Yaskawa INFORM job: OK_R2_O7,1(P)(180,90)OKKR.JBI

/JOB
//NAME OK_R2_O7,1(P)(180,90)OKKR
///FOLDERNAME X4
//POS
///NPOS 170,170,170,10,0,0
///TOOL 0
///POSTYPE PULSE
///PULSE
C00000=-124821,-99493,-112304,-12763,69065,-63689
C00001=-125572,-109805,-73016,-14673,60245,-62954
C00002=-125529,-106474,-67472,-14933,58606,-62713
C00003=-125513,-105112,-65225,-15043,57949,-62613
C00004=-125931,-102761,-62431,-15024,57379,-62697
C00005=-125513,-105112,-65225,-15043,57949,-62613
C00006=-115155,-116372,-68286,-18066,56230,-58210
C00007=-113191,-117815,-68179,-18629,55880,-57359
C00008=-115155,-116372,-68286,-18066,56230,-58210
C00009=-115178,-117983,-70589,-17944,56786,-58316
C00010=-115234,-121991,-76286,-17657,58155,-58571
C00011=-120585,-128453,-93269,-11576,67473,-62203
C00012=-120088,-125588,-88095,-11803,65866,-61858
C00013=-119888,-124404,-86000,-11898,65228,-61718
C00014=-120403,-122095,-83389,-11849,64741,-61858
C00015=-119888,-124404,-86000,-11898,65228,-61718
C00016=-108971,-134765,-87218,-14096,62473,-57335
C00017=-106536,-136286,-87094,-14543,62053,-56368
C00018=-108971,-134765,-87218,-14096,62473,-57335
C00019=-109237,-136316,-89410,-13991,62964,-57496
C00020=-109895,-140195,-94852,-13741,64173,-57891
C00021=-125550,-127827,-102093,-6546,69504,-64123
C00022=-124619,-125212,-97090,-6829,67858,-63692
C00023=-124246,-124117,-95064,-6945,67210,-63518
C00024=-124692,-122258,-93043,-6859,66886,-63662
C00025=-124246,-124117,-95064,-6945,67210,-63518
C00026=-116781,-135280,-96410,-8903,63075,-60474
C00027=-115485,-136646,-96399,-9241,62517,-59943
C00028=-116781,-135280,-96410,-8903,63075,-60474
C00029=-117208,-136830,-98557,-8770,63547,-60670
C00030=-118273,-140721,-103898,-8447,64709,-61154
C00031=-124821,-99493,-112304,-12763,69065,-63689
C00032=-107946,-141846,-124280,-39630,59824,-29939
C00033=-109801,-105651,-82130,-40578,68986,-43153
C00034=-114208,-101668,-58675,-42695,64807,-43138
C00035=-119984,-99571,-57689,-39111,62764,-45440
C00036=-120682,-97946,-55361,-39253,61992,-45447
C00037=-120683,-95917,-52962,-39397,61652,-45306
C00038=-120682,-97946,-55361,-39253,61992,-45447
C00039=-120456,-110188,-58493,-40823,58706,-43930
C00040=-120434,-113010,-58717,-41347,57713,-43467
C00041=-120456,-110188,-58493,-40823,58706,-43930
C00042=-119614,-112042,-60852,-40668,59458,-43865
C00043=-117480,-116658,-66680,-40315,61328,-43677
C00044=-118912,-112770,-80088,-37329,68797,-47272
C00045=-120652,-109018,-74647,-37486,66909,-47352
C00046=-121340,-107497,-72445,-37559,66154,-47379
C00047=-121335,-105659,-70425,-37638,65916,-47288
C00048=-121340,-107497,-72445,-37559,66154,-47379
C00049=-119649,-123976,-76874,-39368,62335,-45109
C00050=-119586,-126928,-76972,-39856,61227,-44619
C00051=-119649,-123976,-76874,-39368,62335,-45109
C00052=-118793,-125859,-79136,-39287,63040,-45003
C00053=-116627,-130595,-84751,-39109,64786,-44716
C00054=-118466,-121522,-88777,-40234,61844,-44303
C00055=-120300,-116165,-83095,-40134,60429,-44594
C00056=-121009,-114063,-80811,-40109,59853,-44695
C00057=-121007,-112566,-79277,-40173,59718,-44636
C00058=-121009,-114063,-80811,-40109,59853,-44695
C00059=-120085,-126490,-82623,-42400,56261,-42581
C00060=-120051,-129243,-82840,-42985,55321,-42099
C00061=-120085,-126490,-82623,-42400,56261,-42581
C00062=-119241,-128903,-84937,-42455,56795,-42402
C00063=-117047,-135114,-90707,-42638,58096,-41900
C00064=-109801,-105651,-82130,-40578,68986,-43153
C00065=-122192,-109712,-75470,-6994,72350,-47586
C00066=-120404,-106593,-70167,-7203,70857,-46871
C00067=-119689,-105303,-68015,-7288,70263,-46584
C00068=-119701,-103141,-65704,-7302,69952,-46569
C00069=-119689,-105303,-68015,-7288,70263,-46584
C00070=-121664,-119459,-71492,-7384,64996,-46952
C00071=-121705,-121620,-70662,-7478,63384,-46863
C00072=-121664,-119459,-71492,-7384,64996,-46952
C00073=-122530,-121046,-73712,-7280,65466,-47290
C00074=-124694,-124965,-79200,-7022,66635,-48130
C00075=-123098,-114349,-89377,-6073,92150,-50670
C00076=-121321,-114367,-85375,-5874,89822,-49955
C00077=-120587,-114243,-83719,-5794,88924,-49665
C00078=-120588,-112592,-81737,-5794,88555,-49647
C00079=-120587,-114243,-83719,-5794,88924,-49665
C00080=-120582,-131484,-87781,-5822,82597,-49371
C00081=-120567,-134184,-87056,-5843,80774,-49281
C00082=-120582,-131484,-87781,-5822,82597,-49371
C00083=-121475,-132061,-89612,-5910,83359,-49704
C00084=-123618,-133239,-94082,-6121,85336,-50515
C00085=-122927,-125261,-102860,-5781,84947,-50274
C00086=-121065,-123842,-98350,-5851,83046,-49551
C00087=-120312,-123169,-96506,-5880,82315,-49259
C00088=-120315,-121628,-95025,-5881,82198,-49255
C00089=-120312,-123169,-96506,-5880,82315,-49259
C00090=-120906,-137774,-98641,-5969,76113,-49167
C00091=-120906,-140631,-98437,-6009,74527,-49089
C00092=-120906,-137774,-98641,-5969,76113,-49167
C00093=-121779,-138951,-100636,-5931,76668,-49494
C00094=-123931,-141761,-105561,-5836,78092,-50300
C00095=-120586,-134579,-103358,-4485,83037,-11114
C00096=-120585,-131353,-98423,-4497,81662,-11065
C00097=-122535,-156833,-100738,-4824,60146,-10922
C00098=-120522,-156760,-100374,-5125,60080,-10181
C00099=-120535,-157089,-102253,-5074,61063,-10231
C00100=-122383,-157140,-100927,-4850,60115,-10864
C00101=-120539,-156480,-102582,-5050,61576,-10256
C00102=-120540,-162054,-108025,-5027,62060,-10277
C00103=-120585,-128403,-93705,-30706,64058,-34634
C00104=-120567,-133478,-88916,-33924,55149,-31719
C00105=-122986,-144654,-84100,-43838,39416,-25487
C00106=-120515,-146044,-85731,-44330,40764,-24767
C00107=-120500,-145449,-83725,-45099,40100,-24310
C00108=-106025,-137078,-79844,-52562,53027,-19025
C00109=-92891,-135829,-78811,-56182,61380,-16538
C00110=-84226,-141246,-87089,-54613,67539,-15724
C00111=-120583,-120823,-82153,-31538,61287,-33793
C00112=-120582,-117425,-76976,-31951,60054,-33402
C00113=-121881,-133792,-71539,-46034,38379,-24018
C00114=-120512,-134879,-73160,-46011,39332,-23778
C00115=-120497,-134214,-71093,-46846,38685,-23292
C00116=-121927,-133795,-71532,-46028,38354,-24030
C00117=-120517,-134657,-73586,-45684,39595,-23969
C00118=-120519,-139446,-79120,-44885,40271,-24439
C00119=-120584,-125271,-89201,-16167,69548,-26657
C00120=-120507,-146022,-83749,-22694,42309,-21504
C00121=-122688,-146060,-81853,-22354,40667,-22120
C00122=-120486,-145618,-81276,-23272,41099,-21150
C00123=-120502,-146316,-83328,-22869,41930,-21396
C00124=-122679,-146211,-81883,-22385,40613,-22104
C00125=-120507,-145977,-83749,-22685,42330,-21510
C00126=-120508,-151207,-89253,-22395,42978,-21687
C00127=-120580,-111726,-68534,-21389,53781,-37532
C00128=-127451,-113025,-63775,-15084,47988,-22225
C00129=-127911,-112838,-61925,-15165,46900,-22250
C00130=-127661,-113044,-61494,-15348,46585,-22086
C00131=-127527,-113364,-63423,-15147,47596,-22194
C00132=-128157,-113633,-62740,-8323,46523,-24870
C00133=-127382,-113593,-64507,-8470,47695,-24640
C00134=-127382,-117368,-69886,-8296,49052,-24759
C00135=-120579,-109195,-64459,-33713,55342,-34372
C00136=-120513,-118310,-53934,-51164,35641,-23385
C00137=-121307,-116964,-51688,-51749,34808,-23220
C00138=-120509,-118473,-53470,-51568,35408,-23161
C00139=-120494,-117670,-51270,-52630,34821,-22576
C00140=-120628,-116889,-51668,-51870,35163,-23019
C00141=-120514,-118344,-53933,-51183,35630,-23374
C00142=-102692,-110233,-56027,-52580,57513,-23173
C00143=-107946,-141846,-124280,-39630,59824,-29939
C00144=-124821,-99493,-112304,-12763,69065,-63689
C00145=-120586,-135028,-103405,-1882,87308,19162
C00146=-95049,-154551,-101030,-14337,69428,29511
C00147=-96126,-153925,-99141,-14396,68431,29253
C00148=-94146,-154571,-100597,-14373,69310,29842
C00149=-92471,-153341,-98557,-14446,68990,30473
C00150=-96000,-153530,-99051,-14384,68596,29277
C00151=-95031,-154583,-101021,-14339,69408,29519
C00152=-95039,-160005,-106445,-14291,69943,29450
C00153=-120584,-127627,-92064,-1887,84134,19210
C00154=-95004,-143259,-88720,-14502,67715,29738
C00155=-95339,-142285,-86410,-14590,66766,29741
C00156=-94099,-143241,-88272,-14539,67610,30071
C00157=-92423,-142062,-86207,-14620,67249,30708
C00158=-95266,-142001,-86258,-14586,66826,29758
C00159=-94987,-143283,-88710,-14504,67700,29747
C00160=-94995,-148127,-94108,-14424,68506,29642
C00161=-126729,-131199,-78425,-7859,72324,12803
C00162=-89985,-126930,-79761,-25221,64343,28101
C00163=-102105,-116048,-60730,-25417,55293,25441
C00164=-99787,-132576,-70465,-18596,67244,23022
C00165=-98008,-131339,-68291,-18558,66943,23687
C00166=-115076,-125750,-62730,-24557,48304,21778
C00167=-95026,-148562,-70381,-25080,50029,28750
C00168=-77295,-139943,-72591,-26428,68032,32942
C00169=-120677,-167921,-121518,-9910,88025,13948
BC00000=174963,806561,1075175
BC00001=174963,859467,1075175
BC00002=174963,859467,1075175
BC00003=174963,859467,1075175
BC00004=174963,859467,1075175
BC00005=174963,859467,1075175
BC00006=174963,859467,1075175
BC00007=174963,859467,1075175
BC00008=174963,859467,1075175
BC00009=174963,859467,1075175
BC00010=174963,859467,1075175
BC00011=189251,842480,1075175
BC00012=189251,842480,1075175
BC00013=189251,842480,1075175
BC00014=189251,842480,1075175
BC00015=189251,842480,1075175
BC00016=189251,842480,1075175
BC00017=189251,842480,1075175
BC00018=189251,842480,1075175
BC00019=189251,842480,1075175
BC00020=189251,842480,1075175
BC00021=209854,804511,1075175
BC00022=209854,804511,1075175
BC00023=209854,804511,1075175
BC00024=209854,804511,1075175
BC00025=209854,804511,1075175
BC00026=209854,804511,1075175
BC00027=209854,804511,1075175
BC00028=209854,804511,1075175
BC00029=209854,804511,1075175
BC00030=209854,804511,1075175
BC00031=174963,806561,1075175
BC00032=274409,813354,1075175
BC00033=301256,838628,1075175
BC00034=300201,927123,1075175
BC00035=300201,927123,1075175
BC00036=300201,927123,1075175
BC00037=300201,927123,1075175
BC00038=300201,927123,1075175
BC00039=300201,927123,1075175
BC00040=300201,927123,1075175
BC00041=300201,927123,1075175
BC00042=300201,927123,1075175
BC00043=300201,927123,1075175
BC00044=301479,887201,1075175
BC00045=301479,887201,1075175
BC00046=301479,887201,1075175
BC00047=301479,887201,1075175
BC00048=301479,887201,1075175
BC00049=301479,887201,1075175
BC00050=301479,887201,1075175
BC00051=301479,887201,1075175
BC00052=301479,887201,1075175
BC00053=301479,887201,1075175
BC00054=301256,838628,1075175
BC00055=301256,838628,1075175
BC00056=301256,838628,1075175
BC00057=301256,838628,1075175
BC00058=301256,838628,1075175
BC00059=301256,838628,1075175
BC00060=301256,838628,1075175
BC00061=301256,838628,1075175
BC00062=301256,838628,1075175
BC00063=301256,838628,1075175
BC00064=301256,838628,1075175
BC00065=342983,940837,1075175
BC00066=342983,940837,1075175
BC00067=342983,940837,1075175
BC00068=342983,940837,1075175
BC00069=342983,940837,1075175
BC00070=342983,940837,1075175
BC00071=342983,940837,1075175
BC00072=342983,940837,1075175
BC00073=342983,940837,1075175
BC00074=342983,940837,1075175
BC00075=341951,928188,1075175
BC00076=341951,928188,1075175
BC00077=341951,928188,1075175
BC00078=341951,928188,1075175
BC00079=341951,928188,1075175
BC00080=341951,928188,1075175
BC00081=341951,928188,1075175
BC00082=341951,928188,1075175
BC00083=341951,928188,1075175
BC00084=341951,928188,1075175
BC00085=341833,876223,1075175
BC00086=341833,876223,1075175
BC00087=341833,876223,1075175
BC00088=341833,876223,1075175
BC00089=341833,876223,1075175
BC00090=341833,876223,1075175
BC00091=341833,876223,1075175
BC00092=341833,876223,1075175
BC00093=341833,876223,1075175
BC00094=341833,876223,1075175
BC00095=326648,872548,1075175
BC00096=327339,875123,1075175
BC00097=327615,876153,1075175
BC00098=327615,876153,1075175
BC00099=327615,876153,1075175
BC00100=343543,876201,1075175
BC00101=343266,875171,1075175
BC00102=342576,872596,1075175
BC00103=288239,845332,1075175
BC00104=287541,847903,1075175
BC00105=287262,848931,1075175
BC00106=287262,848931,1075175
BC00107=287262,848931,1075175
BC00108=271334,848883,1075175
BC00109=271613,847855,1075175
BC00110=271613,847855,1075175
BC00111=288137,879825,1075175
BC00112=287440,882396,1075175
BC00113=287161,883424,1075175
BC00114=287161,883424,1075175
BC00115=287161,883424,1075175
BC00116=271233,883376,1075175
BC00117=271512,882348,1075175
BC00118=272210,879777,1075175
BC00119=343580,891466,1075175
BC00120=344270,894040,1075175
BC00121=344546,895069,1075171
BC00122=344547,895070,1075175
BC00123=344547,895070,1075175
BC00124=360474,895118,1075175
BC00125=360198,894088,1075175
BC00126=359508,891513,1075175
BC00127=346836,915420,1075175
BC00128=347526,917995,1075175
BC00129=347803,919025,1075175
BC00130=347803,919025,1075175
BC00131=347803,919025,1075175
BC00132=354009,918467,1075175
BC00133=353458,917448,1075175
BC00134=352078,914901,1075175
BC00135=287933,917208,1075175
BC00136=287235,919779,1075175
BC00137=286956,920807,1075175
BC00138=286956,920807,1075175
BC00139=286956,920807,1075175
BC00140=271028,920759,1075175
BC00141=271307,919731,1075175
BC00142=272005,917160,1075175
BC00143=274409,813354,1075175
BC00144=174963,806561,1075175
BC00145=221551,843736,1075175
BC00146=219316,845269,1075175
BC00147=218422,845882,1075175
BC00148=218422,845882,1075175
BC00149=218422,845882,1075175
BC00150=206253,835971,1075175
BC00151=207147,835358,1075175
BC00152=209382,833826,1075175
BC00153=198513,870087,1075175
BC00154=196278,871620,1075175
BC00155=195383,872233,1075175
BC00156=195383,872233,1075175
BC00157=195383,872233,1075175
BC00158=183214,862322,1075175
BC00159=184108,861709,1075175
BC00160=186343,860177,1075175
BC00161=186413,912658,1075175
BC00162=179451,874735,1075175
BC00163=179451,874735,1075175
BC00164=182574,914172,1075175
BC00165=182574,914172,1075175
BC00166=179451,874735,1075175
BC00167=171501,903829,1075175
BC00168=174243,902747,1075175
BC00169=186413,912658,1075175
EC00000=1596313,309153
EC00001=1596313,309153
EC00002=1596313,309153
EC00003=1596313,309153
EC00004=1596313,309153
EC00005=1596313,309153
EC00006=1596313,309153
EC00007=1596313,309153
EC00008=1596313,309153
EC00009=1596313,309153
EC00010=1596313,309153
EC00011=1596313,309153
EC00012=1596313,309153
EC00013=1596313,309153
EC00014=1596313,309153
EC00015=1596313,309153
EC00016=1596313,309153
EC00017=1596313,309153
EC00018=1596313,309153
EC00019=1596313,309153
EC00020=1596313,309153
EC00021=1596313,309153
EC00022=1596313,309153
EC00023=1596313,309153
EC00024=1596313,309153
EC00025=1596313,309153
EC00026=1596313,309153
EC00027=1596313,309153
EC00028=1596313,309153
EC00029=1596313,309153
EC00030=1596313,309153
EC00031=1596313,309153
EC00032=1596313,556475
EC00033=1596313,556475
EC00034=1596313,556475
EC00035=1596313,556475
EC00036=1596313,556475
EC00037=1596313,556475
EC00038=1596313,556475
EC00039=1596313,556475
EC00040=1596313,556475
EC00041=1596313,556475
EC00042=1596313,556475
EC00043=1596313,556475
EC00044=1596313,556475
EC00045=1596313,556475
EC00046=1596313,556475
EC00047=1596313,556475
EC00048=1596313,556475
EC00049=1596313,556475
EC00050=1596313,556475
EC00051=1596313,556475
EC00052=1596313,556475
EC00053=1596313,556475
EC00054=1596313,556475
EC00055=1596313,556475
EC00056=1596313,556475
EC00057=1596313,556475
EC00058=1596313,556475
EC00059=1596313,556475
EC00060=1596313,556475
EC00061=1596313,556475
EC00062=1596313,556475
EC00063=1596313,556475
EC00064=1596313,556475
EC00065=1596313,556475
EC00066=1596313,556475
EC00067=1596313,556475
EC00068=1596313,556475
EC00069=1596313,556475
EC00070=1596313,556475
EC00071=1596313,556475
EC00072=1596313,556475
EC00073=1596313,556475
EC00074=1596313,556475
EC00075=1596313,556475
EC00076=1596313,556475
EC00077=1596313,556475
EC00078=1596313,556475
EC00079=1596313,556475
EC00080=1596313,556475
EC00081=1596313,556475
EC00082=1596313,556475
EC00083=1596313,556475
EC00084=1596313,556475
EC00085=1596313,556475
EC00086=1596313,556475
EC00087=1596313,556475
EC00088=1596313,556475
EC00089=1596313,556475
EC00090=1596313,556475
EC00091=1596313,556475
EC00092=1596313,556475
EC00093=1596313,556475
EC00094=1596313,556475
EC00095=1596313,556475
EC00096=1596313,556475
EC00097=1596313,556475
EC00098=1596313,556475
EC00099=1596313,556475
EC00100=1596313,556475
EC00101=1596313,556475
EC00102=1596313,556475
EC00103=1596313,556475
EC00104=1596313,556475
EC00105=1596313,556475
EC00106=1596313,556475
EC00107=1596313,556475
EC00108=1596313,556475
EC00109=1596313,556475
EC00110=1596313,556475
EC00111=1596313,556475
EC00112=1596313,556475
EC00113=1596313,556475
EC00114=1596313,556475
EC00115=1596313,556475
EC00116=1596313,556475
EC00117=1596313,556475
EC00118=1596313,556475
EC00119=1596313,556475
EC00120=1596313,556475
EC00121=1596313,556475
EC00122=1596313,556475
EC00123=1596313,556475
EC00124=1596313,556475
EC00125=1596313,556475
EC00126=1596313,556475
EC00127=1596313,556475
EC00128=1596313,556475
EC00129=1596313,556475
EC00130=1596313,556475
EC00131=1596313,556475
EC00132=1596313,556475
EC00133=1596313,556475
EC00134=1596313,556475
EC00135=1596313,556475
EC00136=1596313,556475
EC00137=1596313,556475
EC00138=1596313,556475
EC00139=1596313,556475
EC00140=1596313,556475
EC00141=1596313,556475
EC00142=1596313,556475
EC00143=1596313,556475
EC00144=1596313,309153
EC00145=1596313,309153
EC00146=1596313,309153
EC00147=1596313,309153
EC00148=1596313,309153
EC00149=1596313,309153
EC00150=1596313,309153
EC00151=1596313,309153
EC00152=1596313,309153
EC00153=1596313,309153
EC00154=1596313,309153
EC00155=1596313,309153
EC00156=1596313,309153
EC00157=1596313,309153
EC00158=1596313,309153
EC00159=1596313,309153
EC00160=1596313,309153
EC00161=1596313,309153
EC00162=1596313,309153
EC00163=1596313,309153
EC00164=1596313,309153
EC00165=1596313,309153
EC00166=1596313,309153
EC00167=1596313,309153
EC00168=1596313,309153
EC00169=1596313,309153
///POSTYPE BASE
///RECTAN
///RCONF 0,0,0,0,0,0,0,0,0,0,0,0,0,0,0,0,0,0,0,0,0,0,0,0
P00006=0.222,-3.123,-1.508,0.0000,0.0000,0.0000
P00021=-0.225,-6.128,-0.405,0.0000,0.0000,0.0000
P00022=0.222,-3.123,-1.508,0.0000,0.0000,0.0000
P00023=0.143,-0.036,0.682,0.0000,0.0000,0.0000
P00031=1.853,-0.001,-1.549,0.0000,0.0000,0.0000
P00032=1.957,0.503,-7.217,0.0000,0.0000,0.0000
///RCONF 0,0,0,0,1,0,0,0,0,0,0,0,0,0,0,0,0,0,0,0,0,0,0,0
P00033=-0.123,0.612,-5.012,0.0000,0.0000,0.0000
///RCONF 0,0,0,0,0,0,0,0,0,0,0,0,0,0,0,0,0,0,0,0,0,0,0,0
P00034=-0.304,0.773,-2.693,0.0000,0.0000,0.0000
P00035=2.817,0.591,-1.622,0.0000,0.0000,0.0000
P00036=-1.108,-0.829,1.850,0.0000,0.0000,0.0000
//INST
///DATE 2023/12/13 11:22
///ATTR SC,RW
///GROUP1 RB1,BS1
///GROUP2 ST1
NOP
'OK_r2_O7.1(P)(180,90)
'180,50
MOVJ C00000 BC00000 VJ=100.00  +MOVJ EC00000 VJ=100.00
'Path S1422
SFTOF3D
MOVJ C00001 BC00001 VJ=100.00  +MOVJ EC00001 VJ=100.00
MOVL C00002 BC00002 V=400.0  +MOVJ EC00002 VJ=100.00
SMOVL C00003 BC00003 V=60.0  +MOVJ EC00003
SREFP 3 C00004 BC00004  +REFP EC00004
CALL JOB:SEARCH-R1-S13D
SET P021 P006
SFTON3D P021
SMOVL C00005 BC00005 V=60.0  +MOVJ EC00005
SMOVL C00006 BC00006 V=60.0  +MOVJ EC00006
SREFP 3 C00007 BC00007  +REFP EC00007
CALL JOB:SEARCH-R1-S13D
SET P021 P006
SFTON3D P021
SMOVL C00008 BC00008 V=60.0  +MOVJ EC00008
MOVL C00009 BC00009 V=400.0  +MOVJ EC00009 VJ=100.00
MOVL C00010 BC00010 V=1000.0  +MOVJ EC00010 VJ=100.00
'Path S1423
SFTOF3D
MOVJ C00011 BC00011 VJ=100.00  +MOVJ EC00011 VJ=100.00
MOVL C00012 BC00012 V=400.0  +MOVJ EC00012 VJ=100.00
SMOVL C00013 BC00013 V=60.0  +MOVJ EC00013
SREFP 3 C00014 BC00014  +REFP EC00014
CALL JOB:SEARCH-R1-S13D
SET P022 P006
SFTON3D P022
SMOVL C00015 BC00015 V=60.0  +MOVJ EC00015
SMOVL C00016 BC00016 V=60.0  +MOVJ EC00016
SREFP 3 C00017 BC00017  +REFP EC00017
CALL JOB:SEARCH-R1-S13D
SET P022 P006
SFTON3D P022
SMOVL C00018 BC00018 V=60.0  +MOVJ EC00018
MOVL C00019 BC00019 V=400.0  +MOVJ EC00019 VJ=100.00
MOVL C00020 BC00020 V=1000.0  +MOVJ EC00020 VJ=100.00
'Path S1424
SFTOF3D
MOVJ C00021 BC00021 VJ=100.00  +MOVJ EC00021 VJ=100.00
MOVL C00022 BC00022 V=400.0  +MOVJ EC00022 VJ=100.00
SMOVL C00023 BC00023 V=60.0  +MOVJ EC00023
SREFP 3 C00024 BC00024  +REFP EC00024
CALL JOB:SEARCH-R1-S13D
SET P023 P006
SFTON3D P023
SMOVL C00025 BC00025 V=60.0  +MOVJ EC00025
SMOVL C00026 BC00026 V=60.0  +MOVJ EC00026
SREFP 3 C00027 BC00027  +REFP EC00027
CALL JOB:SEARCH-R1-S13D
SET P023 P006
SFTON3D P023
SMOVL C00028 BC00028 V=60.0  +MOVJ EC00028
MOVL C00029 BC00029 V=400.0  +MOVJ EC00029 VJ=100.00
MOVL C00030 BC00030 V=1000.0  +MOVJ EC00030 VJ=100.00
MOVJ C00031 BC00031 VJ=100.00  +MOVJ EC00031 VJ=100.00
MOVJ C00032 BC00032 VJ=100.00  +MOVJ EC00032 VJ=100.00
'180,0
MOVJ C00033 BC00033 VJ=100.00  +MOVJ EC00033 VJ=100.00
'Path S1077
SFTOF3D
MOVJ C00034 BC00034 VJ=100.00  +MOVJ EC00034 VJ=100.00
MOVL C00035 BC00035 V=400.0  +MOVJ EC00035 VJ=100.00
SMOVL C00036 BC00036 V=60.0  +MOVJ EC00036
SREFP 3 C00037 BC00037  +REFP EC00037
CALL JOB:SEARCH-R1-S13D
SET P031 P006
SFTON3D P031
SMOVL C00038 BC00038 V=60.0  +MOVJ EC00038
SMOVL C00039 BC00039 V=60.0  +MOVJ EC00039
SREFP 3 C00040 BC00040  +REFP EC00040
CALL JOB:SEARCH-R1-S13D
SET P031 P006
SFTON3D P031
SMOVL C00041 BC00041 V=60.0  +MOVJ EC00041
MOVL C00042 BC00042 V=400.0  +MOVJ EC00042 VJ=100.00
MOVL C00043 BC00043 V=1000.0  +MOVJ EC00043 VJ=100.00
'Path S1078
SFTOF3D
MOVJ C00044 BC00044 VJ=100.00  +MOVJ EC00044 VJ=100.00
MOVL C00045 BC00045 V=400.0  +MOVJ EC00045 VJ=100.00
SMOVL C00046 BC00046 V=60.0  +MOVJ EC00046
SREFP 3 C00047 BC00047  +REFP EC00047
CALL JOB:SEARCH-R1-S13D
SET P032 P006
SFTON3D P032
SMOVL C00048 BC00048 V=60.0  +MOVJ EC00048
SMOVL C00049 BC00049 V=60.0  +MOVJ EC00049
SREFP 3 C00050 BC00050  +REFP EC00050
CALL JOB:SEARCH-R1-S13D
SET P032 P006
SFTON3D P032
SMOVL C00051 BC00051 V=60.0  +MOVJ EC00051
MOVL C00052 BC00052 V=400.0  +MOVJ EC00052 VJ=100.00
MOVL C00053 BC00053 V=1000.0  +MOVJ EC00053 VJ=100.00
'Path S1079
SFTOF3D
MOVJ C00054 BC00054 VJ=100.00  +MOVJ EC00054 VJ=100.00
MOVL C00055 BC00055 V=400.0  +MOVJ EC00055 VJ=100.00
SMOVL C00056 BC00056 V=60.0  +MOVJ EC00056
SREFP 3 C00057 BC00057  +REFP EC00057
CALL JOB:SEARCH-R1-S13D
SET P033 P006
SFTON3D P033
SMOVL C00058 BC00058 V=60.0  +MOVJ EC00058
SMOVL C00059 BC00059 V=60.0  +MOVJ EC00059
SREFP 3 C00060 BC00060  +REFP EC00060
CALL JOB:SEARCH-R1-S13D
SET P033 P006
SFTON3D P033
SMOVL C00061 BC00061 V=60.0  +MOVJ EC00061
MOVL C00062 BC00062 V=400.0  +MOVJ EC00062 VJ=100.00
MOVL C00063 BC00063 V=1000.0  +MOVJ EC00063 VJ=100.00
MOVJ C00064 BC00064 VJ=100.00  +MOVJ EC00064 VJ=100.00
'Path S1080
SFTOF3D
MOVJ C00065 BC00065 VJ=100.00  +MOVJ EC00065 VJ=100.00
MOVL C00066 BC00066 V=400.0  +MOVJ EC00066 VJ=100.00
SMOVL C00067 BC00067 V=60.0  +MOVJ EC00067
SREFP 3 C00068 BC00068  +REFP EC00068
CALL JOB:SEARCH-R1-S13D
SET P034 P006
SFTON3D P034
SMOVL C00069 BC00069 V=60.0  +MOVJ EC00069
SMOVL C00070 BC00070 V=60.0  +MOVJ EC00070
SREFP 3 C00071 BC00071  +REFP EC00071
CALL JOB:SEARCH-R1-S13D
SET P034 P006
SFTON3D P034
SMOVL C00072 BC00072 V=60.0  +MOVJ EC00072
MOVL C00073 BC00073 V=400.0  +MOVJ EC00073 VJ=100.00
MOVL C00074 BC00074 V=1000.0  +MOVJ EC00074 VJ=100.00
'Path S1081
SFTOF3D
MOVJ C00075 BC00075 VJ=100.00  +MOVJ EC00075 VJ=100.00
MOVL C00076 BC00076 V=400.0  +MOVJ EC00076 VJ=100.00
SMOVL C00077 BC00077 V=60.0  +MOVJ EC00077
SREFP 3 C00078 BC00078  +REFP EC00078
CALL JOB:SEARCH-R1-S13D
SET P035 P006
SFTON3D P035
SMOVL C00079 BC00079 V=60.0  +MOVJ EC00079
SMOVL C00080 BC00080 V=60.0  +MOVJ EC00080
SREFP 3 C00081 BC00081  +REFP EC00081
CALL JOB:SEARCH-R1-S13D
SET P035 P006
SFTON3D P035
SMOVL C00082 BC00082 V=60.0  +MOVJ EC00082
MOVL C00083 BC00083 V=400.0  +MOVJ EC00083 VJ=100.00
MOVL C00084 BC00084 V=1000.0  +MOVJ EC00084 VJ=100.00
'Path S1082
SFTOF3D
MOVJ C00085 BC00085 VJ=100.00  +MOVJ EC00085 VJ=100.00
MOVL C00086 BC00086 V=400.0  +MOVJ EC00086 VJ=100.00
SMOVL C00087 BC00087 V=60.0  +MOVJ EC00087
SREFP 3 C00088 BC00088  +REFP EC00088
CALL JOB:SEARCH-R1-S13D
SET P036 P006
SFTON3D P036
SMOVL C00089 BC00089 V=60.0  +MOVJ EC00089
SMOVL C00090 BC00090 V=60.0  +MOVJ EC00090
SREFP 3 C00091 BC00091  +REFP EC00091
CALL JOB:SEARCH-R1-S13D
SET P036 P006
SFTON3D P036
SMOVL C00092 BC00092 V=60.0  +MOVJ EC00092
MOVL C00093 BC00093 V=400.0  +MOVJ EC00093 VJ=100.00
MOVL C00094 BC00094 V=1000.0  +MOVJ EC00094 VJ=100.00
'Path W260
SFTOF3D
PAUSE
SFTON3D P036
MOVJ C00095 BC00095 VJ=100.00  +MOVJ EC00095 VJ=100.00
SMOVL C00096 BC00096 V=400.0  +MOVJ EC00096
SMOVL C00097 BC00097 V=100.0 PL=0  +MOVJ EC00097
SREFP 1 C00098 BC00098  +REFP EC00098
SREFP 2 C00099 BC00099  +REFP EC00099
MACRO1 MJ#(0) ARGF0
ARCON
SMOVL C00100 BC00100 V=10.0  +MOVJ EC00100
ARCOF
SMOVL C00101 BC00101 V=400.0  +MOVJ EC00101
SMOVL C00102 BC00102 V=1000.0  +MOVJ EC00102
SFTOF3D
'Path W261
SFTOF3D
SFTON3D P033
MOVJ C00103 BC00103 VJ=100.00  +MOVJ EC00103 VJ=100.00
SMOVL C00104 BC00104 V=400.0  +MOVJ EC00104
SMOVL C00105 BC00105 V=100.0 PL=0  +MOVJ EC00105
SREFP 1 C00106 BC00106  +REFP EC00106
SREFP 2 C00107 BC00107  +REFP EC00107
MACRO1 MJ#(0) ARGF0
ARCON
SMOVL C00108 BC00108 V=10.0  +MOVJ EC00108
ARCOF
SMOVL C00109 BC00109 V=400.0  +MOVJ EC00109
SMOVL C00110 BC00110 V=1000.0  +MOVJ EC00110
SFTOF3D
'Path W1083
SFTOF3D
SFTON3D P032
MOVJ C00111 BC00111 VJ=100.00  +MOVJ EC00111 VJ=100.00
SMOVL C00112 BC00112 V=400.0  +MOVJ EC00112
SMOVL C00113 BC00113 V=100.0 PL=0  +MOVJ EC00113
SREFP 1 C00114 BC00114  +REFP EC00114
SREFP 2 C00115 BC00115  +REFP EC00115
MACRO1 MJ#(0) ARGF0
ARCON
SMOVL C00116 BC00116 V=10.0  +MOVJ EC00116
ARCOF
SMOVL C00117 BC00117 V=400.0  +MOVJ EC00117
SMOVL C00118 BC00118 V=1000.0  +MOVJ EC00118
SFTOF3D
'Path W262
SFTOF3D
SFTON3D P035
MOVJ C00119 BC00119 VJ=100.00  +MOVJ EC00119 VJ=100.00
SMOVL C00120 BC00120 V=400.0  +MOVJ EC00120
SMOVL C00121 BC00121 V=100.0 PL=0  +MOVJ EC00121
SREFP 1 C00122 BC00122  +REFP EC00122
SREFP 2 C00123 BC00123  +REFP EC00123
MACRO1 MJ#(0) ARGF0
ARCON
SMOVL C00124 BC00124 V=10.0  +MOVJ EC00124
ARCOF
SMOVL C00125 BC00125 V=400.0  +MOVJ EC00125
SMOVL C00126 BC00126 V=1000.0  +MOVJ EC00126
SFTOF3D
'Path W264
SFTOF3D
SFTON3D P034
MOVJ C00127 BC00127 VJ=100.00  +MOVJ EC00127 VJ=100.00
SMOVL C00128 BC00128 V=400.0  +MOVJ EC00128
SMOVL C00129 BC00129 V=100.0 PL=0  +MOVJ EC00129
SREFP 1 C00130 BC00130  +REFP EC00130
SREFP 2 C00131 BC00131  +REFP EC00131
MACRO1 MJ#(0) ARGF0
ARCON
SMOVL C00132 BC00132 V=10.0  +MOVJ EC00132
ARCOF
SMOVL C00133 BC00133 V=400.0  +MOVJ EC00133
SMOVL C00134 BC00134 V=1000.0  +MOVJ EC00134
SFTOF3D
'Path W263
SFTOF3D
SFTON3D P031
MOVJ C00135 BC00135 VJ=100.00  +MOVJ EC00135 VJ=100.00
SMOVL C00136 BC00136 V=400.0  +MOVJ EC00136
SMOVL C00137 BC00137 V=100.0 PL=0  +MOVJ EC00137
SREFP 1 C00138 BC00138  +REFP EC00138
SREFP 2 C00139 BC00139  +REFP EC00139
MACRO1 MJ#(0) ARGF0
ARCON
SMOVL C00140 BC00140 V=10.0  +MOVJ EC00140
ARCOF
SMOVL C00141 BC00141 V=400.0  +MOVJ EC00141
SMOVL C00142 BC00142 V=1000.0  +MOVJ EC00142
SFTOF3D
MOVJ C00143 BC00143 VJ=100.00  +MOVJ EC00143 VJ=100.00
'180,50
MOVJ C00144 BC00144 VJ=100.00  +MOVJ EC00144 VJ=100.00
'Path W1425
SFTOF3D
PAUSE
SFTON3D P023
MOVJ C00145 BC00145 VJ=100.00  +MOVJ EC00145 VJ=100.00
SMOVL C00146 BC00146 V=100.0  +MOVJ EC00146
SMOVL C00147 BC00147 V=100.0 PL=0  +MOVJ EC00147
SREFP 1 C00148 BC00148  +REFP EC00148
SREFP 2 C00149 BC00149  +REFP EC00149
MACRO1 MJ#(0) ARGF0
ARCON
SMOVL C00150 BC00150 V=10.0  +MOVJ EC00150
ARCOF
SMOVL C00151 BC00151 V=400.0  +MOVJ EC00151
SMOVL C00152 BC00152 V=1000.0  +MOVJ EC00152
SFTOF3D
'Path W1426
SFTOF3D
SFTON3D P022
MOVJ C00153 BC00153 VJ=100.00  +MOVJ EC00153 VJ=100.00
SMOVL C00154 BC00154 V=100.0  +MOVJ EC00154
SMOVL C00155 BC00155 V=100.0 PL=0  +MOVJ EC00155
SREFP 1 C00156 BC00156  +REFP EC00156
SREFP 2 C00157 BC00157  +REFP EC00157
MACRO1 MJ#(0) ARGF0
ARCON
SMOVL C00158 BC00158 V=10.0  +MOVJ EC00158
ARCOF
SMOVL C00159 BC00159 V=400.0  +MOVJ EC00159
SMOVL C00160 BC00160 V=1000.0  +MOVJ EC00160
SFTOF3D
'Path W1427
SFTOF3D
SFTON3D P021
MOVJ C00161 BC00161 VJ=100.00  +MOVJ EC00161 VJ=100.00
SMOVL C00162 BC00162 V=100.0  +MOVJ EC00162
SMOVL C00163 BC00163 V=100.0 PL=0  +MOVJ EC00163
SREFP 1 C00164 BC00164  +REFP EC00164
SREFP 2 C00165 BC00165  +REFP EC00165
MACRO1 MJ#(0) ARGF0
ARCON
SMOVL C00166 BC00166 V=10.0  +MOVJ EC00166
ARCOF
SMOVL C00167 BC00167 V=400.0  +MOVJ EC00167
SMOVL C00168 BC00168 V=1000.0  +MOVJ EC00168
SFTOF3D
MOVJ C00169 BC00169 VJ=100.00  +MOVJ EC00169 VJ=100.00
END
